(* PLC project v0.6.04_CycleSemiAuto.project, CODESYS CODESYS V3.5 SP19 Patch 1 *)
(* stored: creationDateTime 2026-07-23T21:30:34.014397, modificationDateTime 2026-07-23T21:30:34.014397 *)

(* ═══════════════════════════════════════════════════════════════ 🎮 ST_SyncCmd — Commandes IHM pour la synchronisation M1/M2 ═══════════════════════════════════════════════════════════════ *)
TYPE ST_SyncCmd : STRUCT
  SelSyncEnable : BOOL := TRUE;  (* ☑️ coché = synchro voulue (MAINT_N1/N2), ex-OverrideSync inversé *)
END_STRUCT;
END_TYPE
